(* IEC 61131-3 sources: control/src, 5 files *)

(* ---- IController.st ---- *)
NAMESPACE Simatic.Ax.Control
    INTERFACE IController
        METHOD Calculate : LREAL
        END_METHOD
    END_INTERFACE
END_NAMESPACE

(* ---- ITimeprovider.st ---- *)
NAMESPACE Simatic.Ax.Control

    INTERFACE ITimeProvider
        /// Returns the time base in ms
        METHOD GetTime : LREAL
        END_METHOD
    END_INTERFACE

    CLASS TimeProviderFixedTimeBase
        IMPLEMENTS ITimeProvider
        VAR PUBLIC
            TimeBase : LREAL := 10;
        END_VAR

        METHOD PUBLIC GetTime : LREAL
            GetTime := TimeBase;
        END_METHOD
    END_CLASS

END_NAMESPACE

(* ---- Controller.st ---- *)
NAMESPACE Simatic.Ax.Control

    CLASS D_Controller EXTENDS ControllerAbstract

        METHOD PROTECTED OVERRIDE _calculate : LREAL
            VAR
                error : LREAL;
            END_VAR
            IF (TimeBase = NULL) THEN
                RETURN;
            END_IF;
            error := SetpointValue - ActualValue^;
            _errorSum := _errorSum + error;
            _calculate := Kp * Td / TimeBase.GetTime() * (error - _errorPre);
            _errorPre := error;
        END_METHOD
    END_CLASS

    CLASS PI_Controller EXTENDS ControllerAbstract

        METHOD PROTECTED OVERRIDE _calculate : LREAL
            VAR
                error : LREAL;
            END_VAR
            IF (TimeBase = NULL) THEN
                RETURN;
            END_IF;
            error := SetpointValue - ActualValue^;
            _errorSum := _errorSum + error;
            _calculate := Kp * error + Kp * TimeBase.GetTime() / Tn * _errorSum;
            _errorPre := error;
        END_METHOD
    END_CLASS

    CLASS PIDController EXTENDS ControllerAbstract

        METHOD PROTECTED OVERRIDE _calculate : LREAL
            VAR
                error : LREAL;
            END_VAR
            VAR_TEMP
                _timebase : LREAL;
            END_VAR
            IF (TimeBase = NULL) THEN
                RETURN;
            END_IF;
            _timebase := TimeBase.GetTime();
            error := SetpointValue - ActualValue^;
            _errorSum := _errorSum + error;
            _calculate := Kp * error + Kp * _timebase / Tn * _errorSum + Kp * Td / _timebase * (error - _errorPre);
            _errorPre := error;
        END_METHOD

    END_CLASS

END_NAMESPACE

(* ---- ControllerAbstract.st ---- *)
NAMESPACE Simatic.Ax.Control

    CLASS ABSTRACT ControllerAbstract
        IMPLEMENTS IController
        VAR PUBLIC
            Kp : LREAL;
            Tn : LREAL;
            Td : LREAL;
            TimeBase : ITimeProvider;
            SetpointValue : LREAL;
            ActualValue : REF_TO LREAL;
        END_VAR
        VAR PROTECTED
            _errorPre : LREAL;
            _errorSum : LREAL;
            _statusError : BOOL;
        END_VAR

        /// method which has to be called cyclically
        METHOD PUBLIC Calculate : LREAL
            _statusError := NOT (THIS.Check());
            IF (_statusError) THEN
                RETURN;
            ELSE
                Calculate := THIS._calculate();
            END_IF;
        END_METHOD

        /// Abstract method: must be implemented in the concrete controller type
        METHOD PROTECTED ABSTRACT _calculate : LREAL
        END_METHOD

        METHOD PROTECTED Check : BOOL
            Check := (TimeBase <> NULL) AND (ActualValue <> NULL);
        END_METHOD
    END_CLASS

END_NAMESPACE

(* ---- myClass.st ---- *)
NAMESPACE Simatic.Ax.Library

    {axcode:docs-v0:@simatic-ax/control:MyClass.md}
    CLASS MyClass

        VAR PUBLIC
        END_VAR

        VAR
        END_VAR

        /// Inline Comment for MyMethod. It will be shown, when you hover over the method
        /// This method has no parameters and no return value
        METHOD PUBLIC MyMethod
            ;
        END_METHOD

    END_CLASS

END_NAMESPACE
